// TIA Portal V16 export
// export: Created 2021-11-12T13:33:23.103767Z, ExportSetting WithDefaults, DisplayName Totally Integrated Automation Portal, DisplayVersion V16 Update 3, DisplayName TIA Portal Version Control Interface, DisplayVersion V16 Update 2, DisplayName TIA Portal Openness, DisplayVersion V16 Update 3, DisplayName SINAMICS Startdrive Advanced, DisplayVersion V16 Update 5, DisplayName SINAMICS Startdrive G130, G150, S120, S150, SINAMICS MV, S210, DisplayVersion V16 Update 5, DisplayName SINAMICS Startdrive G110M, G120, G120C, G120D, G120P, G115D, DisplayVersion V16 Update 5, DisplayName STEP 7 Professional, DisplayVersion V16 Update 3, DisplayName STEP 7 Safety, DisplayVersion V16, DisplayName WinCC UA Professional, DisplayVersion V16 Update 3
DATA_BLOCK "UserDiag_HmiData"   // DB21003
{ S7_Optimized_Access := 'TRUE' }
VERSION : 0.1
// stored: AutoNumber false, DBAccessibleFromOPCUA true, InstanceOfName UserDiag_typeHmiData, InstanceOfType UDT, IsOnlyStoredInLoadMemory false, IsWriteProtectedInAS false
"UserDiag_typeHmiData"
   // VAR
   //    actIOSystem : Int;
   //    actDeviceOfScreen : Int;
   //    ioSlotDiagnosticsLoaded : Bool;
   //    actScreenDevices : Int;
   //    maxScreensDevices : Int;
   //    ackWaitTime : Int;
   //    ackStates : Bool;
   //    actIOSystemData { S7_SetPoint := 'True'} : "UserDiag_typeActIOSystem";
   //    actDeviceNumber : UInt;
   //    actDeviceName : String[50];
   //    actIPAddress { S7_SetPoint := 'True'} : IP_V4;
   //    errorAtLowerScreen : Bool;
   //    errorAtUpperScreen : Bool;
   //    filterErrorDevices : Bool;
   //    ioSystemError : Array[1.."USERDIAG_IO_SYSTEMS_UPPER_LIM"] of Bool;
   // END_VAR
BEGIN
END_DATA_BLOCK
